{region '#Template'}
	{attribute 'Version' := '5.0.0.0'}
	{attribute 'Tags' := '"LCID": "1031", "Text": "Universal, Pump"'}
	{attribute 'Tags' := '"LCID": "1033", "Text": "Universal, Pump"'}
	{attribute 'Using' := '"Type": "Template", "URI": "EC_ID"'}
	{attribute 'Using' := '"Type": "Template", "URI": "BA2_Param"'}
	{attribute 'Description' := '"LCID": "1031", "Text": "Pumpe 1 stufig"'}
	{attribute 'Description' := '"LCID": "1033", "Text": "Pump 1 stage"'}
{endregion}	 
FUNCTION_BLOCK FB_BA_Pu1st EXTENDS FB_BA_Mot1st
VAR_INPUT
	bAblkLock				: BOOL;	
END_VAR
VAR_INPUT CONSTANT
	DlyOff					: FB_BA_DlyOff;								
	Ablk					: FB_BA_AntiBlocking;							
END_VAR
VAR
	PrioSwiPgm				: FB_BA_PrioSwi_B04;
	tonAblkLock				: TON;
END_VAR
VAR // added by the converter: edge detectors and wires of the graphical bodies
    _s1 : ST_BA_Binary;
END_VAR

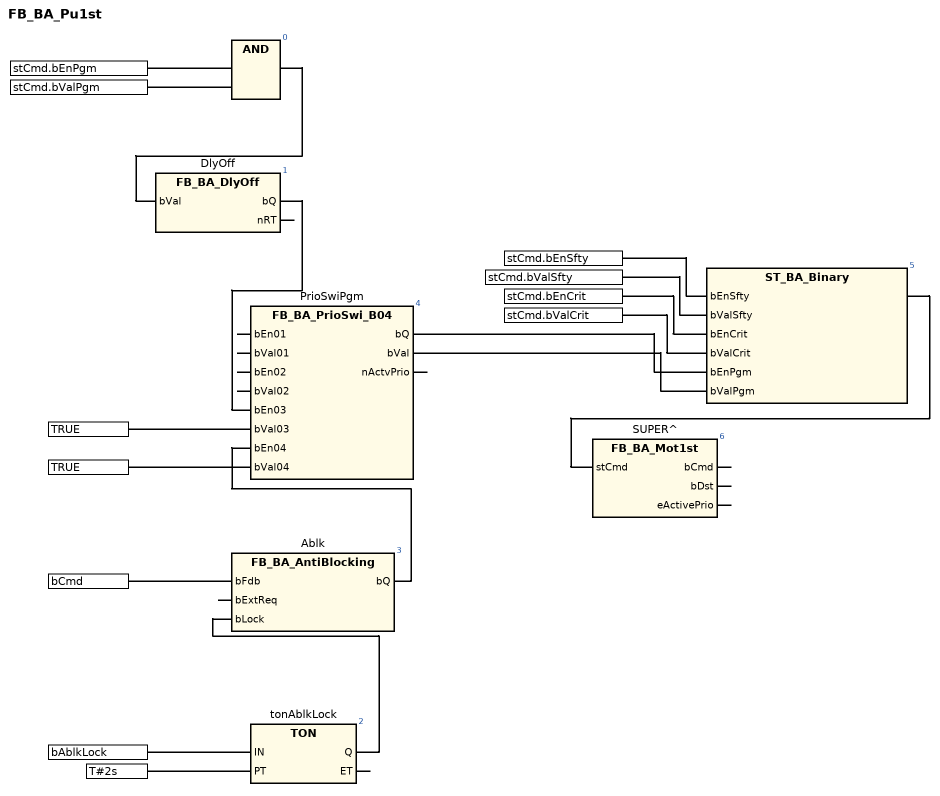
DlyOff(bVal := stCmd.bEnPgm AND stCmd.bValPgm); // FB_BA_DlyOff
tonAblkLock(IN := bAblkLock, PT := T#2s); // TON
Ablk(bFdb := bCmd, bLock := tonAblkLock.Q); // FB_BA_AntiBlocking
PrioSwiPgm(bEn03 := DlyOff.bQ, bVal03 := TRUE, bEn04 := Ablk.bQ, bVal04 := TRUE); // FB_BA_PrioSwi_B04
// compose _s1 : ST_BA_Binary
_s1.bEnSfty := stCmd.bEnSfty;
_s1.bValSfty := stCmd.bValSfty;
_s1.bEnCrit := stCmd.bEnCrit;
_s1.bValCrit := stCmd.bValCrit;
_s1.bEnPgm := PrioSwiPgm.bQ;
_s1.bValPgm := PrioSwiPgm.bVal;
SUPER^(stCmd := _s1); // FB_BA_Mot1st

METHOD FB_init : BOOL
VAR_INPUT
	bInitRetains : BOOL; // if TRUE, the retain variables are initialized (warm start / cold start)
	bInCopyCode : BOOL;  // if TRUE, the instance afterwards gets moved into the copy code (online change)
END_VAR
DlyOff.iParent			:= THIS^;	
DlyOff.iLabel			:= LblCtl_DelayOff;
DlyOff.eDPADMode		:= E_BA_DPADMode.eIncludeDescription;

Ablk.iParent			:= THIS^;	 
Ablk.iLabel				:= LblCtl_AntiBlocking;
Ablk.eDPADMode			:= E_BA_DPADMode.eIncludeDescription;
END_METHOD

END_FUNCTION_BLOCK

(* stored: Version 1.1.0.1, ProductVersion 3.1.4024.12
   POU FB_BA_Pu1st: Id {cb61a7ab-c855-4cf8-9120-2a34d3597527}, SpecialFunc None
   Method FB_init: Id {8ab03f2e-99d0-40d4-ae99-798d8cb41cef} *)
